// TIA Portal V20 export
TYPE "CBS_Carrier"
   STRUCT
      Carrier_Cargado : Bool;   // A true indica que está cargado, a false vacío
      vagon_cargado_SinDestino : Bool;   // Indica que tiene una carga pero que no se le ha asignado destino para la misma
      carrier_no_utilizable : Bool;   // Indica que el vagón está defectuoso y que no se puede utilizar
      vagon_reservado_carga : Bool;   // Indica que el vagón va a ser utilizado para cargar desde un punto concreto
      carrier_multiple : Bool;   // Indica que el vagón es múltiple
      Reserva_5 : Bool;
      Reserva_6 : Bool;
      Reserva_7 : Bool;
      Reserva_8 : Bool;
      Reserva_9 : Bool;
      Reserva_10 : Bool;
      Reserva_11 : Bool;
      Reserva_12 : Bool;
      Reserva_13 : Bool;
      Reserva_14 : Bool;
      Reserva_15 : Bool;
      numero_vagon : UInt;   // Indica el número de vagón del que se trata dentro del sorter
      punto_entrada_carga : UInt;   // Número identificativo de la entrada que ha cargado el vagón
      Destino_principal : Int;   // Numero identificativo del destino principal
      Destino_alternativo : Int;   // Numero identificativo del destino secundario
      Mesa_descarga : Int;
      Num_Recirculaciones : Int;   // cantidad de recirculaciones que ha tenido el vagón cargado
      Numero_Vagones_Multiple_Asociados : Int;   // Cantidad de carriers que tiene asociados formando el vagón multiple
      EventoAGenerar : UInt;
      DatosCarga : Struct   // Datos de la Carga
         Mckey : UDInt;   // Mckey
         MesaOrigen : UInt;   // MesaOrigen
         MesaDestino : UInt;   // MesaDestino
         EtiquetaRouter : UDInt;   // Etiqueta
      END_STRUCT;
   END_STRUCT;
END_TYPE
